FUNCTION_BLOCK DataPanel_xDB0808_DIO_SAE_J1939 (* Service Interface Function Block Type *)
  (* Standard: SAE J1939; Function: Combo Block: 8 Inputs/8 Outputs (includes all input/output types); Type: DP-34044-1-000; Description: this maps to IX/QX *)
  (* Version 1.0, 2018-12-05, Jose Cabral *)
  (* Version 1.1, 2022-08-04, Franz Höpfinger, HR Agrartechnik GmbH *)
  (* Version 1.2, 2023-01-05, Franz Höpfinger, HR Agrartechnik GmbH *)
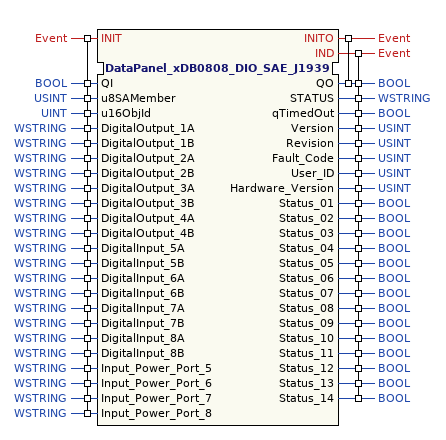
  EVENT_INPUT
    INIT WITH QI, u8SAMember, u16ObjId, DigitalOutput_1A, DigitalOutput_1B, DigitalOutput_2A, DigitalOutput_2B, DigitalOutput_3A, DigitalOutput_3B, DigitalOutput_4A, DigitalOutput_4B, DigitalInput_5A, DigitalInput_5B, DigitalInput_7A, DigitalInput_6A, DigitalInput_6B, DigitalInput_7B, DigitalInput_8A, DigitalInput_8B, Input_Power_Port_5, Input_Power_Port_6, Input_Power_Port_7, Input_Power_Port_8; (* Service Initialization *)
  END_EVENT
  EVENT_OUTPUT
    INITO WITH QO; (* Initialization Confirm *)
    IND WITH QO, STATUS, qTimedOut, Version, Revision, Fault_Code, User_ID, Hardware_Version, Status_01, Status_02, Status_03, Status_04, Status_05, Status_06, Status_07, Status_08, Status_09, Status_10, Status_11, Status_12, Status_13, Status_14; (* Indication from Resource *)
  END_EVENT
  VAR_INPUT
    QI : BOOL; (* Event Input Qualifier *)
    u8SAMember : USINT := 224; (* Node SA 224..239 *)
    u16ObjId : UINT := 65535; (* Dummy ! set to 65535 if in Doubt. 0 deactivates FB. *)
    DigitalOutput_1A : WSTRING := "DigitalOutput_1A";
    DigitalOutput_1B : WSTRING := "DigitalOutput_1B";
    DigitalOutput_2A : WSTRING := "DigitalOutput_2A";
    DigitalOutput_2B : WSTRING := "DigitalOutput_2B";
    DigitalOutput_3A : WSTRING := "DigitalOutput_3A";
    DigitalOutput_3B : WSTRING := "DigitalOutput_3B";
    DigitalOutput_4A : WSTRING := "DigitalOutput_4A";
    DigitalOutput_4B : WSTRING := "DigitalOutput_4B";
    DigitalInput_5A : WSTRING := "DigitalInput_5A";
    DigitalInput_5B : WSTRING := "DigitalInput_5B";
    DigitalInput_6A : WSTRING := "DigitalInput_6A";
    DigitalInput_6B : WSTRING := "DigitalInput_6B";
    DigitalInput_7A : WSTRING := "DigitalInput_7A";
    DigitalInput_7B : WSTRING := "DigitalInput_7B";
    DigitalInput_8A : WSTRING := "DigitalInput_8A";
    DigitalInput_8B : WSTRING := "DigitalInput_8B";
    Input_Power_Port_5 : WSTRING := "Input_Power_Port_5";
    Input_Power_Port_6 : WSTRING := "Input_Power_Port_6";
    Input_Power_Port_7 : WSTRING := "Input_Power_Port_7";
    Input_Power_Port_8 : WSTRING := "Input_Power_Port_8";
  END_VAR
  VAR_OUTPUT
    QO : BOOL; (* Event Output Qualifier *)
    STATUS : WSTRING; (* Service Status *)
    qTimedOut : BOOL;
    Version : USINT;
    Revision : USINT;
    Fault_Code : USINT;
    User_ID : USINT;
    Hardware_Version : USINT;
    Status_01 : BOOL;
    Status_02 : BOOL;
    Status_03 : BOOL;
    Status_04 : BOOL;
    Status_05 : BOOL;
    Status_06 : BOOL;
    Status_07 : BOOL;
    Status_08 : BOOL;
    Status_09 : BOOL;
    Status_10 : BOOL;
    Status_11 : BOOL;
    Status_12 : BOOL;
    Status_13 : BOOL;
    Status_14 : BOOL;
  END_VAR
END_FUNCTION_BLOCK
